// TIA Portal V16 export
// export: Created 2025-10-06T17:54:34.0902688Z, ExportSetting WithDefaults, DisplayName Totally Integrated Automation Portal, DisplayVersion V16, DisplayName TIA Portal Version Control Interface, DisplayVersion V16, DisplayName TIA Portal Openness, DisplayVersion V16, DisplayName STEP 7 Professional, DisplayVersion V16, DisplayName STEP 7 Safety, DisplayVersion V16, DisplayName WinCC Advanced, DisplayVersion V16
DATA_BLOCK "PLCMemory"   // DB15
VERSION : 0.1
// stored: AutoNumber true, IsOnlyStoredInLoadMemory false, IsWriteProtectedInAS false
   VAR RETAIN
      Homing_Sensor_Wals_Offset_Test : Time := T#1S_200MS;   // Offset of homing position sensor wals
      Wals_Delay_Offset : Time := T#400MS;   // Offset of Wals on delay
      Safety_Delay : Time := T#5MS;   // Delay of safety high
      WalsCheck_Time : Time := T#5S;   // Time offset when wals slipping message is displayed
      ProductCheck_Time : Time := T#15S;   // Time offset when aanvoer not in position message is displayed
      ProductIntervalTime : Time := T#10s;   // Counts the time between 2 products
      ProductIntervalTime_1 : Time;   // Depends on ProductIntervalTimer
      ProductIntervalTime_2 : Time;   // Depends on ProductIntervalTimer_1
      TD_Products_Counter : Int;   // Counts the total amount of products with the Sensor Band
      UsernameMemory : String := 'Key';
      PasswordMemory : String := 'Key123';
      SpeedSettingsTakeover : Bool := True;   // Makes the speed of Overname the same as speed Drive 1
      SpeedSettingOvername : Bool;   // Parameter of setting the speed for Drive 4 (Overname)
      SpeedSettingBand : Bool;   // Parameter of setting the speed for Drive 1 (Band)
      TimingSettingOvername : Bool := True;   // Makes the timing of Overname the same as speed Drive 1
      EncoderPosition : Real;   // Real Value of Encoder Axis 3 (Wals)
      StepSize : Real := 0.0;   // Pulsfactor of Encoder Axis 3
      Desired_Encoder_Position : Real;
      Tolerance : Real := 0.0;
      "Encoder PulsOffset" : Time := T#3MS;
      Axis3_Ref_Pos : Real := 85.0;   // Refention position of Axis 3 without tolerance
      Reference_Position_Axis3 : Real;   // Refention position of Axis 3 with calculated tolerance
      ProductCount : Int;
      Axis3_ControlMode : Bool := true;
      Axis1_ControlMode : Bool := true;
      ProductsToProduce : Int;
      SystemTime : Time;
      Disable_Modules : Struct
         Disable_Band : Bool;
         Disable_Trilgoten : Bool;
         Disable_AanvoerWals : Bool;
         Disable_Aandruk1 : Bool;
         Disable_Aandruk2 : Bool;
         Disable_Aandruk3 : Bool;
         Disable_Blaaspuls : Bool;
         Disable_Retourband : Bool;
         Disable_Afsluiter : Bool;
      END_STRUCT;
      Offset_Timers : Struct
         Trilgoten_Start_Offset : Time := T#10MS;   // Delay offset of start trilgoten
         Trilgoten_Stop_Offset : Time := T#10MS;   // Delay offset of stop trilgoten
         Aanvoer_Start_Offset : Time := T#10MS;   // Delay offset of start aanvoer
         Magazijn_Sensor_Delay : Time := T#15S;   // Delay on magazijn sensor.
         Aanvoer_Stop_Offset : Time := T#10MS;   // Delay offset of stop aanvoer
         Overname_Start_Offset : Time := T#5MS;   // Delay offset of start Overname
         Overname_Stop_Offset : Time := T#5MS;   // Delay offset of stop Overname
         Retourband_Start_Offset : Time := T#5ms;
         Retourband_Stop_Offset : Time := T#5ms;
         BlowOff_CycleTime : Time := T#500ms;
         Blow_Off_PulseTime : Time := T#500ms;
      END_STRUCT;
      ProductBuffer : Struct
         DelayTime : Time := T#7s;
         ProductsCount : Int;
         MoveTrigger : Bool;
         MoveFeedback : Bool;
         RestFeedback : Bool;
         InsertIndex : Int;
      END_STRUCT;
      ProductBufferBehindWals : Struct
         DelayTime : Time := T#1s_890MS;
         Product_Count : Int;
      END_STRUCT;
      ProductBuffer_1 : Struct
         DelayTime : Time := T#7s;
         ProductsCount : Int;
         MoveTrigger : Bool;
         MoveFeedback : Bool;
         RestFeedback : Bool;
         InsertIndex : Int;
      END_STRUCT;
      TriggerDistanceBand : DInt := 418000;
      TriggerDistanceAandruk : DInt := 500000;
      InfeedTimeOutPT : Time := T#2S;
      "Blow Off Timer on" : Time := T#2S;
      ResetManual : Bool;
   END_VAR
BEGIN
END_DATA_BLOCK
